GLOBALCONSTANTS logiBUS_AI (* logiBUS_DI constants *)
  (* Standard: 61499-1; Description: Copyright (c) 2024 HR Agrartechnik GmbH This program and the accompanying materials are made available under the terms of the Eclipse Public License 2.0 which is available at https://www.eclipse.org/legal/epl-2.0/ SPDX-License-Identifier: EPL-2.0 *)
  (* Version 1.0, 2024-01-25, Franz Höpfinger, HR Agrartechnik GmbH *)
  PACKAGE logiBUS::io::AI;
  IMPORT eclipse4diac::core::TypeHash;
  VAR_GLOBAL CONSTANT
    AnalogInput_I1 : logiBUS::io::AI::logiBUS_AI_S := (Pin := 1);
    AnalogInput_I2 : logiBUS::io::AI::logiBUS_AI_S := (Pin := 2);
    AnalogInput_I3 : logiBUS::io::AI::logiBUS_AI_S := (Pin := 3);
    AnalogInput_I4 : logiBUS::io::AI::logiBUS_AI_S := (Pin := 4);
    AnalogInput_I5 : logiBUS::io::AI::logiBUS_AI_S := (Pin := 5);
    AnalogInput_I6 : logiBUS::io::AI::logiBUS_AI_S := (Pin := 6);
    AnalogInput_I7 : logiBUS::io::AI::logiBUS_AI_S := (Pin := 7);
    AnalogInput_I8 : logiBUS::io::AI::logiBUS_AI_S := (Pin := 8);
    AnalogInput_I9 : logiBUS::io::AI::logiBUS_AI_S := (Pin := 9);
    Invalid : logiBUS::io::AI::logiBUS_AI_S := (Pin := 255);
  END_VAR
END_GLOBALCONSTANTS
